{attribute 'pack_mode' := '0'}
TYPE receive_data_format :
STRUCT
	command		: STRING(4);
	seq_number	: UINT;
	value		: REAL;
END_STRUCT
END_TYPE

(* stored: Version 1.1.0.1, ProductVersion 3.1.4024.12
   DUT receive_data_format: Id {7fbfe23e-69bf-4008-adde-196134391bf0} *)
